KUKA KRL program: module1.src, module1.dat

--- module1.src ---
&ACCESS RVP
&REL 1
&COMMENT New program
DEF module1()
  ;FOLD INI
    ;FOLD BASISTECH INI
      BAS(#INITMOV, 0)
    ;ENDFOLD
  ;ENDFOLD

  PTP HOME Vel=100% DEFAULT

  ; TODO: Add motion commands here

  PTP HOME Vel=100% DEFAULT

END

--- module1.dat ---
DEFDAT module1
  ;FOLD EXTERNAL DECLARATIONS; %{PE}
  ;ENDFOLD

  DECL E6POS HOME={A1 0.0, A2 -90.0, A3 90.0, A4 0.0, A5 0.0, A6 0.0}

ENDDAT
